FUNCTION_BLOCK LSC_TransferWorkpieceTo_RampEnd EXTENDS LSC_MoveWorkpiece_Base
VAR_INPUT
END_VAR
VAR_OUTPUT
END_VAR
VAR
	// EProcessVariables.LSC_WPAtRampEnd = FALSE
	m_precondition: ComparisonExpression(EProcessVariables.LSC_WPAtRampEnd, EComparisonType.equals, EDataType.binary, FALSE, 0, '', TRUE);
	
	// TRUE
	m_postcondition: ValueExpression(EDataType.binary, TRUE, 0, '', TRUE);
END_VAR

SUPER^();

METHOD PROTECTED  AtTarget : BOOL
VAR_INPUT
END_VAR
AtTarget := m_ptrLSC^.WPAtRampEnd;
END_METHOD

METHOD PROTECTED EjectOperation : BOOL
VAR_INPUT
END_VAR
EjectOperation := TRUE;
END_METHOD

METHOD FB_init : BOOL
VAR_INPUT
	bInitRetains : BOOL; // if TRUE, the retain variables are initialized (warm start / cold start)
	bInCopyCode : BOOL;  // if TRUE, the instance afterwards gets moved into the copy code (online change)
	
	i_ptrLSC: POINTER TO LargeSortingConveyor;
END_VAR
m_ptrLSC := i_ptrLSC;

m_id := EPrimitives.LSC_TransferWorkpieceTo_RampEnd;
m_timeout := T#200S;

Precondition := m_precondition;
Postcondition := m_postcondition;
END_METHOD

END_FUNCTION_BLOCK

(* stored: Version 1.1.0.1, ProductVersion 3.1.4024.9
   POU LSC_TransferWorkpieceTo_RampEnd: Id {e519c17d-8231-438d-acfe-c6acd6537afd}, SpecialFunc None
   Method AtTarget: Id {92c5009f-5902-4eaa-9d4d-3931ab643924}
   Method EjectOperation: Id {1ab1e47d-ab28-43d4-8b4e-8055dee4e538}
   Method FB_init: Id {175dac2a-e373-4bfa-9a81-0bc015aafe36} *)
